// TIA Portal V16 export
// export: Created 2022-01-12T14:34:25.9616392Z, ExportSetting WithDefaults, DisplayName Totally Integrated Automation Portal, DisplayVersion V16 Update 4, DisplayName TIA Portal Version Control Interface, DisplayVersion V16 Update 2, DisplayName TIA Portal Openness, DisplayVersion V16 Update 4, DisplayName STEP 7 Professional, DisplayVersion V16 Update 4, DisplayName STEP 7 Safety, DisplayVersion V16, DisplayName WinCC Professional, DisplayVersion V16 Update 4
TYPE "typButton"
// stored: IsFailsafeCompliant false
   STRUCT
      set : Bool;
      reset : Bool;
      widoczny : Bool := 1;
      kolor : Int := 4;
      aktywny : Bool := 1;
   END_STRUCT;
END_TYPE
